FUNCTION_BLOCK ABSTRACT FB_AbstractObserver IMPLEMENTS I_Observer
VAR
END_VAR

{attribute 'hasanytype'}
METHOD ABSTRACT Update : I_Observer
VAR_INPUT
    anyVal:         ANY;
END_VAR
END_METHOD

END_FUNCTION_BLOCK

(* stored: Version 1.1.0.1, ProductVersion 3.1.4024.12
   POU FB_AbstractObserver: Id {59366400-b2f5-4598-9c5c-2530302a1d7f}, SpecialFunc None
   Method Update: Id {db1aebf2-fca2-494e-a52a-f9c476d5cd33} *)
